(* IEC 61131-3 sources: POMIRTS_lab3/AS/Library/AsNxAsiM, 3 files *)

(* ---- AsNxAsiM.typ ---- *)
(********************************************************************
 * COPYRIGHT -- Bernecker + Rainer
 ********************************************************************
 * Library: AsNxAsiM
 * File: AsNxAsiM.typ
 * Author: B+R
 ********************************************************************
 * Data types of library AsNxAsiM
 ********************************************************************)

TYPE
	asimSlaveList_t			: STRUCT				(*slave list*)
		slaveBits			: ARRAY[0..7] OF USINT;	(*slave bits*)
	END_STRUCT;

	asimSlaveDiagnosis_t	: STRUCT				(*slave diagnosis*)
		diagnosisFlags		: UDINT;				(*diagnosis flags*)
		numOfDiagInfos		: UDINT;				(*number of diagnosis infos*)
		slaveError			: ARRAY[0..7] OF UDINT;	(*slave error*)
	END_STRUCT;
END_TYPE

(* ---- AsNxAsiM.fun ---- *)
(********************************************************************
 * COPYRIGHT -- Bernecker + Rainer
 ********************************************************************
 * Library: AsNxAsiM
 * File: AsNxAsiM.fun
 * Author: B+R
 ********************************************************************
 * Functions and function blocks of library AsNxAsiM
 ********************************************************************)

FUNCTION_BLOCK asimWriteParameter			(*write parameter*)
	VAR_INPUT
		enable				: BOOL;			(*enables execution*)
		pDevice				: UDINT;		(*interface name given as a pointer, e.g., "SL<x>.SS<y>.IF<z>"*)
		slaveAddress		: UDINT;		(*slave address*)
		parameterData		: UDINT;		(*parameter data*)
	END_VAR
	VAR
        _state				: UINT;			(*internal variable*)
		_result				: UINT;			(*internal variable*)
        _srcId				: UDINT;		(*internal variable*)
	END_VAR
	VAR_OUTPUT
		status				: UINT;			(*execution status: ERR_OK, ERR_FUB_ENABLE_FALSE, ERR_FUB_BUSY, 0xXXXX = see help*)
		asiStatus			: UDINT;		(*ASI stack status*)
		parameterDataEcho	: UDINT;		(*parameter data echo*)
	END_VAR
END_FUNCTION_BLOCK

FUNCTION_BLOCK asimChangeSlaveAddress	(*change slave address*)
	VAR_INPUT
		enable			: BOOL;			(*enables execution*)
		pDevice			: UDINT;		(*interface name given as a pointer, e.g., "SL<x>.SS<y>.IF<z>"*)
		oldSlaveAddress	: UDINT;		(*old slave address*)
		newSlaveAddress	: UDINT;		(*new slave address*)
	END_VAR
	VAR
        _state			: UINT;			(*internal variable*)
		_result			: UINT;			(*internal variable*)
        _srcId			: UDINT;		(*internal variable*)
	END_VAR
	VAR_OUTPUT
		status			: UINT;			(*execution status: ERR_OK, ERR_FUB_ENABLE_FALSE, ERR_FUB_BUSY, 0xXXXX = see help*)
		asiStatus		: UDINT;		(*ASI stack status*)
	END_VAR
END_FUNCTION_BLOCK

FUNCTION_BLOCK asimGetProjectedSlaves	(*get list of projected slaves*)
	VAR_INPUT
		enable			: BOOL;			(*enables execution*)
		pDevice			: UDINT;		(*interface name given as a pointer, e.g., "SL<x>.SS<y>.IF<z>"*)
		pSlaveList		: UDINT;		(*slave list given as a pointer*)
		maxSlaveListLen	: UDINT;		(*max slave list length*)
	END_VAR
	VAR
        _state			: UINT;			(*internal variable*)
		_result			: UINT;			(*internal variable*)
        _srcId			: UDINT;		(*internal variable*)
	END_VAR
	VAR_OUTPUT
		status			: UINT;			(*execution status: ERR_OK, ERR_FUB_ENABLE_FALSE, ERR_FUB_BUSY, 0xXXXX = see help*)
		asiStatus		: UDINT;		(*ASI stack status*)
		slaveListLen	: UDINT;		(*slave list length*)
	END_VAR
END_FUNCTION_BLOCK

FUNCTION_BLOCK asimGetActivatedSlaves	(*get list of activated slaves*)
	VAR_INPUT
		enable			: BOOL;			(*enables execution*)
		pDevice			: UDINT;		(*interface name given as a pointer, e.g., "SL<x>.SS<y>.IF<z>"*)
		pSlaveList		: UDINT;		(*slave list given as a pointer*)
		maxSlaveListLen	: UDINT;		(*max slave list length*)
	END_VAR
	VAR
        _state			: UINT;			(*internal variable*)
		_result			: UINT;			(*internal variable*)
        _srcId			: UDINT;		(*internal variable*)
	END_VAR
	VAR_OUTPUT
		status			: UINT;			(*execution status: ERR_OK, ERR_FUB_ENABLE_FALSE, ERR_FUB_BUSY, 0xXXXX = see help*)
		asiStatus		: UDINT;		(*ASI stack status*)
		slaveListLen	: UDINT;		(*slave list length*)
	END_VAR
END_FUNCTION_BLOCK

FUNCTION_BLOCK asimGetDetectedSlaves	(*get list of detected slaves*)
	VAR_INPUT
		enable			: BOOL;			(*enables execution*)
		pDevice			: UDINT;		(*interface name given as a pointer, e.g., "SL<x>.SS<y>.IF<z>"*)
		pSlaveList		: UDINT;		(*slave list given as a pointer*)
		maxSlaveListLen	: UDINT;		(*max slave list length*)
	END_VAR
	VAR
        _state			: UINT;			(*internal variable*)
		_result			: UINT;			(*internal variable*)
        _srcId			: UDINT;		(*internal variable*)
	END_VAR
	VAR_OUTPUT
		status			: UINT;			(*execution status: ERR_OK, ERR_FUB_ENABLE_FALSE, ERR_FUB_BUSY, 0xXXXX = see help*)
		asiStatus		: UDINT;		(*ASI stack status*)
		slaveListLen	: UDINT;		(*slave list length*)
	END_VAR
END_FUNCTION_BLOCK

FUNCTION_BLOCK asimGetPeripheralFaults	(*get list of peripheral faults*)
	VAR_INPUT
		enable			: BOOL;			(*enables execution*)
		pDevice			: UDINT;		(*interface name given as a pointer, e.g., "SL<x>.SS<y>.IF<z>"*)
		pSlaveList		: UDINT;		(*slave list given as a pointer*)
		maxSlaveListLen	: UDINT;		(*max slave list length*)
	END_VAR
	VAR
        _state			: UINT;			(*internal variable*)
		_result			: UINT;			(*internal variable*)
        _srcId			: UDINT;		(*internal variable*)
	END_VAR
	VAR_OUTPUT
		status			: UINT;			(*execution status: ERR_OK, ERR_FUB_ENABLE_FALSE, ERR_FUB_BUSY, 0xXXXX = see help*)
		asiStatus		: UDINT;		(*ASI stack status*)
		slaveListLen	: UDINT;		(*slave list length*)
	END_VAR
END_FUNCTION_BLOCK

FUNCTION_BLOCK asimGetSlaveDiagnosis	(*get slave diagnosis*)
	VAR_INPUT
		enable			: BOOL;			(*enables execution*)
		pDevice			: UDINT;		(*interface name given as a pointer, e.g., "SL<x>.SS<y>.IF<z>"*)
		slaveAddress	: UDINT;		(*slave address*)
		requestFlags	: UDINT;		(*request flags*)
		pSlaveDiagnosis	: UDINT;		(*slave diagnosis given as a pointer*)
	END_VAR
	VAR
        _state			: UINT;			(*internal variable*)
		_result			: UINT;			(*internal variable*)
        _srcId			: UDINT;		(*internal variable*)
	END_VAR
	VAR_OUTPUT
		status			: UINT;			(*execution status: ERR_OK, ERR_FUB_ENABLE_FALSE, ERR_FUB_BUSY, 0xXXXX = see help*)
		asiStatus		: UDINT;		(*ASI stack status*)
	END_VAR
END_FUNCTION_BLOCK

(* ---- AsNxAsiM.var ---- *)
(********************************************************************
 * COPYRIGHT -- Bernecker + Rainer
 ********************************************************************
 * Library: AsNxAsiM
 * File: AsNxAsiM.var
 * Author: B+R
 ********************************************************************
 * Local variables of library AsNxAsiM
 ********************************************************************)

VAR CONSTANT
	asimERR_INVALID_DEVICE				: UINT	:= 35030;	(*error invalid device*)
	asimERR_SEND_MESSAGE				: UINT	:= 35031;	(*error send message*)
	asimERR_TIMEOUT						: UINT	:= 35032;	(*error timeout*)
	asimERR_ASI_STACK					: UINT	:= 35033;	(*error receive message*)
	asimERR_PARAMETER					: UINT	:= 35034;	(*error parameter*)
	asimERR_LENGTH						: UINT	:= 35035;	(*error max length*)

	asimDIAG_REQ_FLAG_PEEK				: UDINT	:= 16#00000001;	(*diagnose request flag peek*)
END_VAR
